// SIMATIC S7-200 project (STEP 7-Micro/WIN), CPU 224XP REL 02.00

SYMBOL_TABLE USR1
Always_On        SM0.0    // This bit is always on.
First_Scan_On    SM0.1    // This bit is on for the first scan cycle only.
Time_0_Intrvl    SMB34    // Specifies time interval (5 ms to 255 ms: 1-ms increment) for timed interrupt 0.
Time_1_Intrvl    SMB35    // Specifies time interval (5 ms to 255 ms: 1-ms increment) for timed interrupt 1.
END_SYMBOL_TABLE

SYMBOL_TABLE 
USS_LOW_V        VD1000
USS_HIGH_V       VD1004
USS_TIME_OUT     VW1008
USS_I_LINE       VW1010
USS_DAT_PTR0     VD1012
USS_ACT_DRV0     VD1016
USS_CUR_DRV0     VD1020
USS_P0           V1024.0
USS_REQ_SNT0     V1024.1
USS_RETRY_P0     VB1025
USS_ERR_CODE     VB1026
USS_CS_D0        VD1027
USS_CS_W0        VW1027
USS_CS_W2        VW1029
USS_CS_B0        VB1027
USS_CS_B1        VB1028
USS_POLL_BUF     VB1031
USS_XMT_0        VB1046
USS_XMT_ADR0     VB1049
USS_X_STWD       VD1056
USS_X_BCC        VB1060
USS_X_DW1        VD1047
USS_X_DW5        VD1051
USS_X_DW9        VD1055
USS_X_DB13       VB1059
USS_RCV_BUF0     VB1061
USS_R_STX        VB1062
USS_R_LGE        VB1063
USS_R_ADR        VB1064
USS_R_STWD       VD1071
USS_R_DW1        VD1062
USS_R_DW5        VD1066
USS_R_DW9        VD1070
USS_R_W13        VW1074
USS_STAT_TAB     VB1076
USS_ADR_P0       VB1396
END_SYMBOL_TABLE

ORGANIZATION_BLOCK MAIN:OB1
TITLE=
//  题目：处理定时中断
// ***概述***
// 本例用定时中断来产生闪烁频率脉冲。当连在输入端IO.1的开关接通时，闪烁频率减半；
// 当连在输入端I0.0的开关接通时，又恢复成原有的闪烁频率。
// 本例叙述由定时中断引起的一般性处理以及改变其时间基准。
// 
// ***程序和注释***
// 用特殊存储字节SMB34指定第一定时中断的时间基准，由此产生的定时中断称为中断事件10。
// 用特殊存储字节SMB35指定第二定时中断的时间基准，由此产生的定时中断称为中断事件11。
// 这两种定时中断的时间基准的设定值只能以1ms(毫秒）为单位增加，允
// 许最小值是5ms,最大值是255ms。本例程序组成如下：
//   Main    主程序        初始化和指定时间基准
//   INT0  中断程序0     对输出Q0.0置位（Q0.0=1)
//   INT1   中断程序1    对输出Q0.0复位（Q0.0=0)
// 标题：定时中断
// 
BEGIN
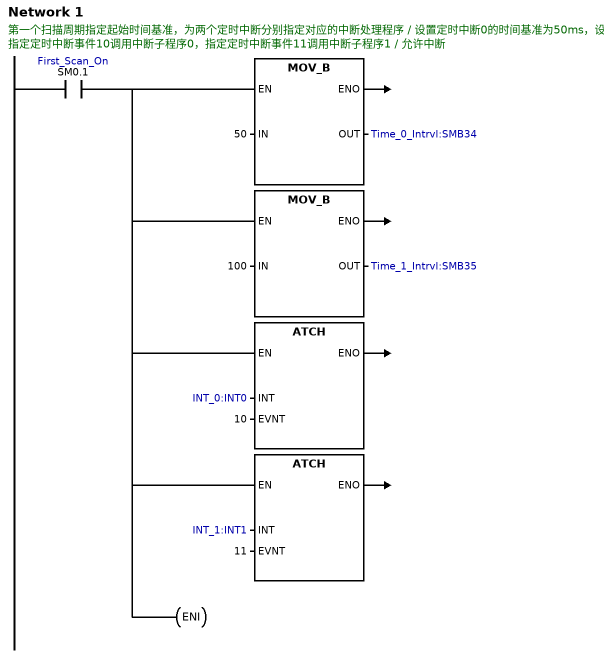
Network 1
// 第一个扫描周期指定起始时间基准，为两个定时中断分别指定对应的中断处理程序
// 设置定时中断0的时间基准为50ms，设置定时中断1的时间基准为100ms
// 指定定时中断事件10调用中断子程序0，指定定时中断事件11调用中断子程序1
// 允许中断
// 仅首次扫描处理
// 设置定时中断0的时间基准为50ms。
// 设置定时中断1的时间基准为100ms。
// 指定定时中断事件10调用中断程序0
// 指定定时中断事件11调用中断程序1
// 允许中断。
LD     First_Scan_On:SM0.1
MOVB   50, Time_0_Intrvl:SMB34
MOVB   100, Time_1_Intrvl:SMB35
ATCH   INT_0:INT0, 10
ATCH   INT_1:INT1, 11
ENI
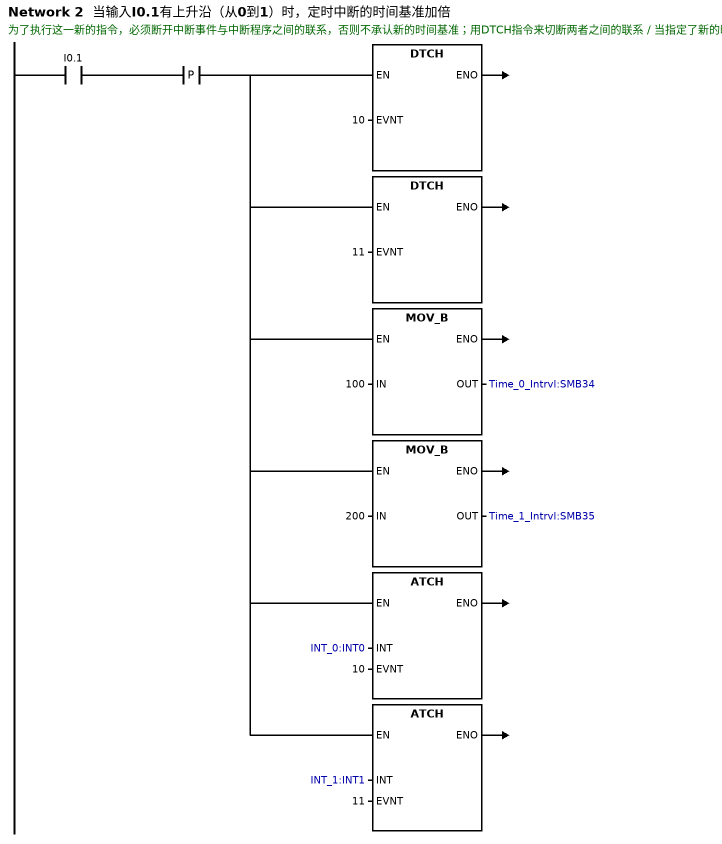
Network 2 // 当输入I0.1有上升沿（从0到1）时，定时中断的时间基准加倍
// 为了执行这一新的指令，必须断开中断事件与中断程序之间的联系，否则不承认新的时间基准；用DTCH指令来切断两者之间的联系
// 当指定了新的时间基准后，必须用ATCH指令来恢复中断事件与中断程序之间的联系
// 输入I0.1
// 上升沿。
// 切断定时中断事件10与中断程序0的联系。
// 切断定时中断事件11与中断程序1的联系。
// 设置定时中断0的新的时间基准为100ms。
// 设置定时中断1的新的时间基准为200ms。
// 恢复定时中断事件10调用中断程序0。
// 恢复定时中断事件11调用中断程序1。
LD     I0.1
EU
DTCH   10
DTCH   11
MOVB   100, Time_0_Intrvl:SMB34
MOVB   200, Time_1_Intrvl:SMB35
ATCH   INT_0:INT0, 10
ATCH   INT_1:INT1, 11
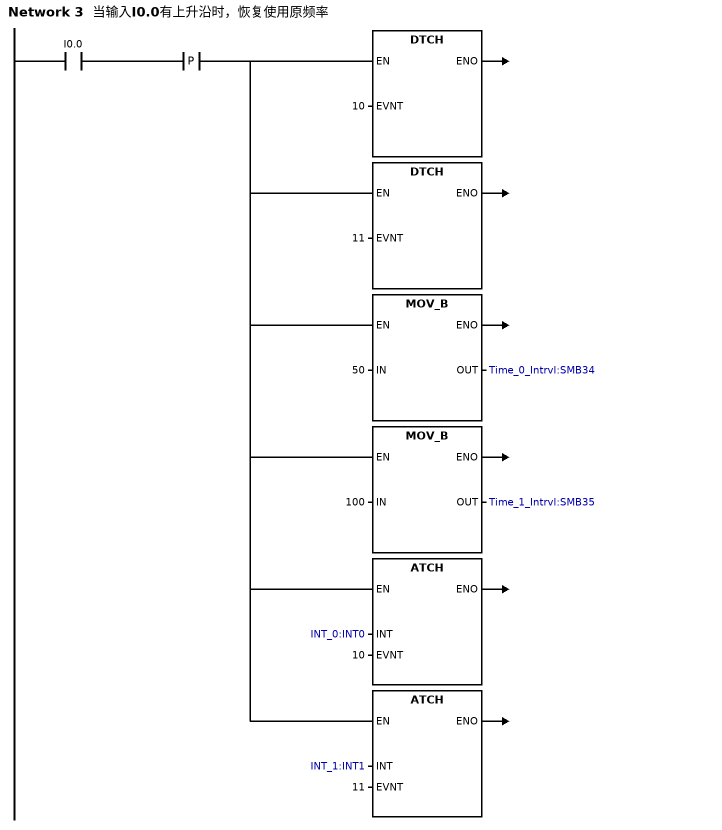
Network 3 // 当输入I0.0有上升沿时，恢复使用原频率
// 输入I0.0
// 上升沿
// 切断定时中断事件10与中断程序0的联系。
// 切断定时中断事件11与中断程序1的联系。
// 设置定时中断0的新的时间基准为50ms。
// 设置定时中断1的新的时间基准为100ms。
// 恢复定时中断事件10与中断程序0的联系。
// 恢复定时中断事件11与中断程序1的联系。
LD     I0.0
EU
DTCH   10
DTCH   11
MOVB   50, Time_0_Intrvl:SMB34
MOVB   100, Time_1_Intrvl:SMB35
ATCH   INT_0:INT0, 10
ATCH   INT_1:INT1, 11
Network 4 //  主程序结束。
//  MEND
// 
END_ORGANIZATION_BLOCK

INTERRUPT_BLOCK INT_0:INT0
TITLE=
BEGIN
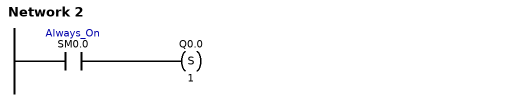
Network 2
//特殊储存器位SM0.0总是1
//把输出Q0.0置位（Q0.0=1）
LD     Always_On:SM0.0
S      Q0.0, 1
Network 3 //  中断程序0结束
//  RETI
// 
END_INTERRUPT_BLOCK

INTERRUPT_BLOCK INT_1:INT1
TITLE=
BEGIN
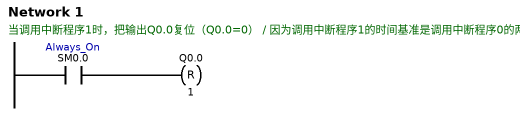
Network 1
// 当调用中断程序1时，把输出Q0.0复位（Q0.0=0）
// 因为调用中断程序1的时间基准是调用中断程序0的两倍，所以输出端Q0.0输出的脉冲频率发生闪烁
// SM0.0总是1
// 把输出Q0.0复位（Q0.0=0）
LD     Always_On:SM0.0
R      Q0.0, 1
Network 2 // 中断程序1结束
//  RETI
// 
END_INTERRUPT_BLOCK
